// TIA Portal project "FillingTank_ControlFunction" (V15)
// This is a test for a control function that doesn´t has a dynamical model, in this case this is going to control the filling of a tank from a factory io scene.

(* hardware
DEVICE "S7-1200 station_1"  S7-1200 Station
   slot 0: "Rack_0"  S7-1200 Rack  Rack  V1.0
   slot 1: "PLC_1"  CPU 1212C AC/DC/Rly  6ES7 212-1BE40-0XB0  V4.2
*)

// ===== PLC "PLC_1"  CPU 1212C AC/DC/Rly =====

VAR_GLOBAL   // PLC tag table "Tabla de variables estándar"
   "Sensor_nivel" AT %EW48 : Int;
END_VAR

DATA_BLOCK "DataBlock_ControlFunction"   // DB2
{ S7_Optimized_Access := 'TRUE' }
VERSION : 0.1
// stored: InstanceOfName ControlFunction
"ControlFunction"
BEGIN
   "B" := 1.0;
END_DATA_BLOCK

// folder: Analog_signals

DATA_BLOCK "Analog_Inputs"   // DB1
{ S7_Optimized_Access := 'TRUE' }
VERSION : 0.1
   VAR
      LevelSensor_Normalization : Real;
      LevelSensor_Measure : Real;
      LevelSensor_Input : Real;
   END_VAR
BEGIN
END_DATA_BLOCK

DATA_BLOCK "Analog_Outputs"   // DB3
{ S7_Optimized_Access := 'TRUE' }
VERSION : 0.1
   VAR
      Analog_Output1 : Real;
      Analog_Output1_Normalized : Real;
      Analog_Output2_Normalized : Real;
      Analog_Output2 : Real;
   END_VAR
BEGIN
END_DATA_BLOCK

// folder: (top level)

ORGANIZATION_BLOCK "Main"   // OB1, LAD, ProgramCycle
TITLE = "Main Program Sweep (Cycle)"
{ S7_Optimized_Access := 'TRUE' }
VERSION : 0.1
   VAR_INPUT
      Initial_Call : Bool;   // Initial call of this OB
      Remanence : Bool;   // =True, if remanent data are available
   END_VAR
BEGIN

REGION Network 1
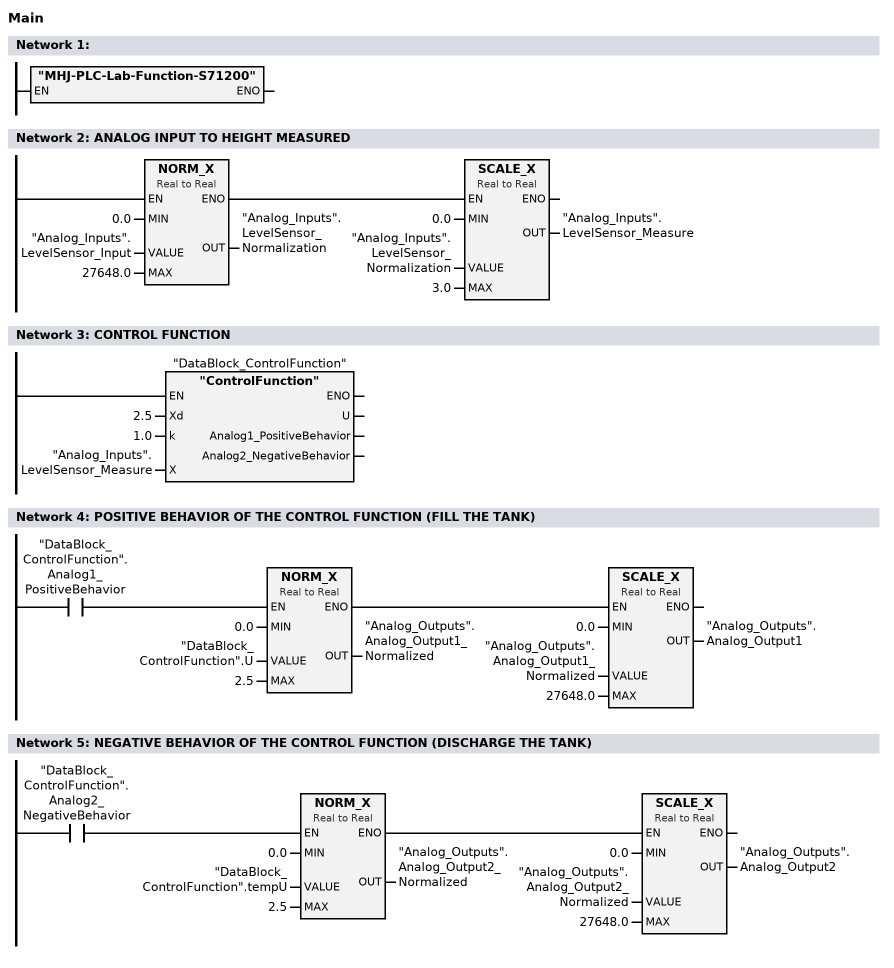
   RUNG wire#powerrail
      "MHJ-PLC-Lab-Function-S71200"()
   END_RUNG
   // the same network as SCL:
   "MHJ-PLC-Lab-Function-S71200"();
END_REGION

REGION Network 2: ANALOG INPUT TO HEIGHT MEASURED
   RUNG wire#powerrail
      { S7_Templates := "[SrcType := Real, DestType := Real]" } Normalize(min := 0.0, value := "Analog_Inputs".LevelSensor_Input, max := 27648.0, out => "Analog_Inputs".LevelSensor_Normalization)
      { S7_Templates := "[SrcType := Real, DestType := Real]" } Scale(min := 0.0, value := "Analog_Inputs".LevelSensor_Normalization, max := 3.0, out => "Analog_Inputs".LevelSensor_Measure)
   END_RUNG
   // the same network as SCL:
   "Analog_Inputs".LevelSensor_Normalization := NORM_X(MIN := 0.0, VALUE := "Analog_Inputs".LevelSensor_Input, MAX := 27648.0);
   "Analog_Inputs".LevelSensor_Measure := SCALE_X(MIN := 0.0, VALUE := "Analog_Inputs".LevelSensor_Normalization, MAX := 3.0);
END_REGION

REGION Network 3: CONTROL FUNCTION
   RUNG wire#powerrail
      "DataBlock_ControlFunction"(Xd := 2.5, k := 1.0, X := "Analog_Inputs".LevelSensor_Measure, U =>, Analog1_PositiveBehavior =>, Analog2_NegativeBehavior =>)
   END_RUNG
   // the same network as SCL:
   "DataBlock_ControlFunction"(Xd := 2.5, k := 1.0, X := "Analog_Inputs".LevelSensor_Measure);   // "ControlFunction"
END_REGION

REGION Network 4: POSITIVE BEHAVIOR OF THE CONTROL FUNCTION (FILL THE TANK)
   RUNG wire#powerrail
      Contact( "DataBlock_ControlFunction".Analog1_PositiveBehavior )
      { S7_Templates := "[SrcType := Real, DestType := Real]" } Normalize(min := 0.0, value := "DataBlock_ControlFunction".U, max := 2.5, out => "Analog_Outputs".Analog_Output1_Normalized)
      { S7_Templates := "[SrcType := Real, DestType := Real]" } Scale(min := 0.0, value := "Analog_Outputs".Analog_Output1_Normalized, max := 27648.0, out => "Analog_Outputs".Analog_Output1)
   END_RUNG
   // the same network as SCL:
   IF "DataBlock_ControlFunction".Analog1_PositiveBehavior THEN
       "Analog_Outputs".Analog_Output1_Normalized := NORM_X(MIN := 0.0, VALUE := "DataBlock_ControlFunction".U, MAX := 2.5);
       "Analog_Outputs".Analog_Output1 := SCALE_X(MIN := 0.0, VALUE := "Analog_Outputs".Analog_Output1_Normalized, MAX := 27648.0);
   END_IF;
END_REGION

REGION Network 5: NEGATIVE BEHAVIOR OF THE CONTROL FUNCTION (DISCHARGE THE TANK)
   RUNG wire#powerrail
      Contact( "DataBlock_ControlFunction".Analog2_NegativeBehavior )
      { S7_Templates := "[SrcType := Real, DestType := Real]" } Normalize(min := 0.0, value := "DataBlock_ControlFunction".tempU, max := 2.5, out => "Analog_Outputs".Analog_Output2_Normalized)
      { S7_Templates := "[SrcType := Real, DestType := Real]" } Scale(min := 0.0, value := "Analog_Outputs".Analog_Output2_Normalized, max := 27648.0, out => "Analog_Outputs".Analog_Output2)
   END_RUNG
   // the same network as SCL:
   IF "DataBlock_ControlFunction".Analog2_NegativeBehavior THEN
       "Analog_Outputs".Analog_Output2_Normalized := NORM_X(MIN := 0.0, VALUE := "DataBlock_ControlFunction".tempU, MAX := 2.5);
       "Analog_Outputs".Analog_Output2 := SCALE_X(MIN := 0.0, VALUE := "Analog_Outputs".Analog_Output2_Normalized, MAX := 27648.0);
   END_IF;
END_REGION
END_ORGANIZATION_BLOCK

// folder: Control_Function

FUNCTION_BLOCK "ControlFunction"   // FB1, LAD
TITLE = FUNCIÓN DE CONTROL PARA SISTEMAS SIN MODELO DINÁMICO
{ S7_Optimized_Access := 'TRUE' }
VERSION : 0.1
// Esta función contiene los parámetros necesarios para realizar el control de casi cualquier sistema dinámico que no puede modelarse por medio de ecuaciones de ninguna forma. 
// 
// Observaciones:
// - El valor k de ganancia puede volverse un arreglo de ganancias en caso de tener dos variables a   medir en el sistema.
// 
// - El valor de B también puede volverse un arreglo que debe contener una diagonal de unos   dependiendo del número de variables a medir en el sistema.
   VAR_INPUT
      Xd : Real;   // Valor deseado a alcanzar (setpoint)
      k : Real;   // Ganancia del sistema
      X : Real;   // Valor medido por sensor (process value)
   END_VAR
   VAR_OUTPUT
      U : Real;   // Valor de salida hacia el actuador
      Analog1_PositiveBehavior : Bool;
      Analog2_NegativeBehavior : Bool;
   END_VAR
   VAR
      ex : Real;   // Error medido en el sistema
      integral_ex : Real;
      "B" : Real;   // Este tiene un valor de 1 por predeterminado
      d : Real;   // Dinámica no modelada
      X_0 : Real;   // Valor inicial del sistema
      tempU : Real;
   END_VAR
BEGIN

REGION Network 1: ----------| ERROR CALCULATION |----------
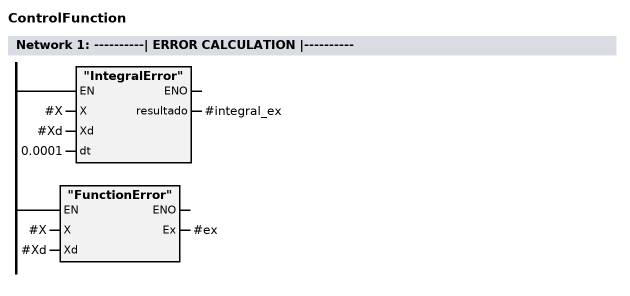
   RUNG wire#powerrail
      "IntegralError"(X := #X, Xd := #Xd, "dt" := 0.0001, resultado => #integral_ex)
   END_RUNG
   RUNG wire#powerrail
      "FunctionError"(X := #X, Xd := #Xd, Ex => #ex)
   END_RUNG
   // the same network as SCL:
   "IntegralError"(X := #X, Xd := #Xd, "dt" := 0.0001, resultado => #integral_ex);
   "FunctionError"(X := #X, Xd := #Xd, Ex => #ex);
END_REGION

REGION Network 2 (SCL): ----------| NON MODELED DYNAMIC |----------
   // d value is stored for the non modeled dynamic
   #d := #X - #X_0-(#B*#k*#integral_ex);
END_REGION

REGION Network 3 (SCL): ----------| INPUT FUNCTION FOR THE SYSTEM |----------
   // The U value can be converted to (0 - 10 V) o (4 - 20 mA) analog signal
   #U := #B * (#k * #ex - #d);
END_REGION

REGION Network 4 (SCL): ----------| CONDITIONS FOR THE INPUT FUNCTION BEHAVIOR |----------
   // - Analog1 works in case the input function gives a postive value
   // 
   // - Analog2 works in case the input function gives a negative value
   // 
   // The two previous variables determined which analog output should work for the system
   IF #U < 0 THEN
       #Analog1_PositiveBehavior := 0;
       #Analog2_NegativeBehavior := 1;
       #tempU := -1 * #U;
   ELSIF #U >= 0 THEN
       #Analog2_NegativeBehavior := 0;
       #Analog1_PositiveBehavior := 1;
   END_IF;
END_REGION
END_FUNCTION_BLOCK

FUNCTION "FunctionError" : Void   // FC2, LAD
TITLE = FUNCIÓN DE ERROR
{ S7_Optimized_Access := 'TRUE' }
VERSION : 0.1
   VAR_INPUT
      X : Real;   // Variable medida desde un sensor analógico (process value)
      Xd : Real;   // Valor deseado (setpoint)
   END_VAR
   VAR_OUTPUT
      Ex : Real;   // Valor del error actual
   END_VAR
BEGIN

REGION Network 1 (SCL): -------------------| CALCULO DEL ERROR |-------------------
   // This function makes the difference between the desired value to reach and the value measured by an analog sensor.
   #Ex := #Xd - #X;
END_REGION
END_FUNCTION

FUNCTION "IntegralError" : Void   // FC3, LAD
TITLE = INTEGRACIÓN DE LA FUNCIÓN DE ERROR
{ S7_Optimized_Access := 'TRUE' }
VERSION : 0.1
// Runge-Kutta 4th order method
   VAR_INPUT
      X : Real;
      Xd : Real;
      "dt" : Real;
   END_VAR
   VAR_OUTPUT
      resultado : Real;   // Integral de la función del error
   END_VAR
   VAR_TEMP
      k1 : Real;   // Valor de la pendiente 1
      k2 : Real;   // Valor de la pendiente 2
      k3 : Real;   // Valor de la pendiente 3
      k4 : Real;   // Valor de la pendiente 4
      df1 : Real;   // Primer diferencial del sistema
      df2 : Real;   // Segundo diferencial del sistema
      df3 : Real;   // Tercer diferencial del sistema
   END_VAR
BEGIN

REGION Network 1: -------------------| SLOPE 1 CALCULATION |-------------------
END_REGION

REGION Network 2 (SCL): Slope 1 value
   "FunctionError"(X:=#X,
                       Xd:=#Xd,
                       Ex=>#k1);
END_REGION

REGION Network 3 (SCL): -------------------| SLOPE 2 CALCULATION |-------------------
END_REGION

REGION Network 4 (SCL): Slope 2 value
   #df1 := 0.5 * #k1 * #dt;

   "FunctionError"(X:=#X+#df1,
                       Xd:=#Xd,
                       Ex=>#k2);
END_REGION

REGION Network 5 (SCL): -------------------| SLOPE 3 CALCULATION |-------------------
END_REGION

REGION Network 6 (SCL): Slope 3 value
   #df2 := 0.5 * #k2 * #dt;

   "FunctionError"(X:=#X+#df2,
                  Xd:=#Xd,
                  Ex=>#k3);
END_REGION

REGION Network 7 (SCL): -------------------| SLOPE 4 CALCULATION |-------------------
END_REGION

REGION Network 8 (SCL): Slope 4 value
   #df3 := #k3 * #dt;

   "FunctionError"(X:=#X+#df3,
                  Xd:=#Xd,
                  Ex=>#k4);
END_REGION

REGION Network 9 (SCL): -------------------| RESULT |-------------------
   #resultado := #X + (#dt / 6) * (#k1 + #k4 + 2 * (#k3 + #k4));
END_REGION
END_FUNCTION

// folder: FactoryIO_connection

FUNCTION "MHJ-PLC-Lab-Function-S71200" : Void   // FC9000, SCL
{ S7_Optimized_Access := 'TRUE' }
VERSION : 0.1
   VAR_TEMP
      rdTimeReturn : Int;
      outputTime : DTL;
      SyncVal : Byte;
      forVal : Int;
      forVal_2 : Int;
      Value : Byte;
   END_VAR
   VAR CONSTANT
      CompVal : Byte := 16#34;
      Value_01 : Byte := 16#11;
      Value_01_DW : DWord := 16#A165_D992;
      Value_02_DW : DWord := 16#58BE_4401;
   END_VAR
BEGIN

   #Value:=PEEK(area := 16#82,
        dbNumber := 0,
        byteOffset := 511);
   #Value := #Value + 1;

   POKE(area := 16#82,
        dbNumber := 0,
        byteOffset := 511,
        value := #Value);

   POKE(area:=16#81,
        dbNumber:=0,
        byteOffset:=1016,
        value:=#Value_01_DW);
   POKE(area := 16#81,
        dbNumber := 0,
        byteOffset := 1020,
        value := #Value_02_DW);

   POKE(area := 16#81,
        dbNumber := 0,
        byteOffset := 511,
        value := B#16#00);

   FOR #forVal := 0 TO 120 DO
       FOR #forVal_2:=0 TO 10 DO
           #rdTimeReturn:=RD_SYS_T(#outputTime);
           #rdTimeReturn := WR_SYS_T(#outputTime);
           #rdTimeReturn := RD_SYS_T(#outputTime);
           #rdTimeReturn := WR_SYS_T(#outputTime);
       END_FOR;
       #SyncVal:= PEEK(area := 16#81,
                      dbNumber := 0,
                      byteOffset := 511);
       IF #SyncVal = #CompVal THEN
          GOTO M_1;
       END_IF;
   END_FOR;
   RETURN;

   M_1:
   POKE(area := 16#81,
        dbNumber := 0,
        byteOffset := 511,
        value := B#16#0);
END_FUNCTION